// TwinCAT 3 PLC project MC3_Multi_IPC2
// ProgramVersion: 3.1.4026.13
// libraries:
//   Tc2_Standard, * (Beckhoff Automation GmbH)
//   Tc2_System, * (Beckhoff Automation GmbH)
//   Tc3_EventLogger, * (Beckhoff Automation GmbH)
//   Tc3_Mc3PlanarMotion, * (Beckhoff Automation GmbH)
//   Tc3_Module, * (Beckhoff Automation GmbH)
//   Tc3_Physics, * (Beckhoff Automation GmbH)
//   Tc3_XL_Motion, * (Beckhoff Automation GmbH)
//   Tc3_XtsInterface,newest,Beckhoff Automation GmbH
// project tree:
//   DUTs/ E_EcState.TcDUT (not stored), E_MergeMode.TcDUT, E_MergeType.TcDUT, E_SwitchOpMode.TcDUT, E_TrackNum.TcDUT, MoverSort.TcDUT, ST_Color_Code.TcDUT (not stored), ST_DataExchange.TcDUT, ST_DivertConfig.TcDUT (not stored), ST_ExchangeData.TcDUT, ST_ExpMoverStatus.TcDUT, ST_MergeConfig.TcDUT (not stored), ST_MoverConfig.TcDUT (not stored), ST_PlanarTrackConfig.TcDUT, ST_SectorConfig.TcDUT, ST_ShortcutConfig.TcDUT, ST_StaticSectorStatus.TcDUT, ST_SwitchConfig.TcDUT (not stored), ST_SwitchStatus.TcDUT, ST_TrackConfig.TcDUT
//   / FB_XtsDataLoggerForController.TcPOU (excluded from build), PlcTask.TcTTO
//   GVLs/ GVL_DataExchange.TcGVL, GVL_MC.TcGVL
//   POUs/ MAIN_S2.TcPOU
//   XlMover/DUTs/ DUT.TcDUT
//   XlMover/ITFs/ I_Mover.TcIO
//   XlMover/POUs/ FB_Mover.TcPOU, F_GetTrackEnum.TcPOU
// (motion and I/O tree: see PLC project saftyplc)
// real-time tasks:
//   TASK XTS Task: cycle T#500us, priority 1, ADS port 350
//   TASK Job Task: cycle default, priority 32
//   TASK MC-Task (MET): cycle T#2ms, priority 3, ADS port 521
//   TASK MC-Task (MPT): cycle T#10ms, priority 8, ADS port 531
//   TASK PlcTask: cycle T#500us, priority 20, ADS port 351
// variable links:
//   MC3_Multi_IPC2/MC3_Multi_IPC2 Instance <-> Device 2 (EtherCAT Automation Protocol)/Box 29 (Subscriber)
//     PlcTask Inputs/GVL_DataExchange.Dynamics <-> Command/Inputs/VarData/Dynamics
//   MC3_Multi_IPC2/MC3_Multi_IPC2 Instance <-> MC Project IPC2/Axes/MC_Mover 01 IPC2
//     PlcTask Inputs/GVL_MC.fbMover[1].fbPlanarMover.MCTOPLC/ACT <-> McToPlc/ACT
//     PlcTask Inputs/GVL_MC.fbMover[1].fbPlanarMover.MCTOPLC/COORDMODE <-> McToPlc/COORDMODE
//     PlcTask Inputs/GVL_MC.fbMover[1].fbPlanarMover.MCTOPLC/SET <-> McToPlc/SET
//     PlcTask Inputs/GVL_MC.fbMover[1].fbPlanarMover.MCTOPLC/SETONTRACK <-> McToPlc/SETONTRACK
//     PlcTask Inputs/GVL_MC.fbMover[1].fbPlanarMover.MCTOPLC/STD <-> McToPlc/STD
//     PlcTask Outputs/GVL_MC.fbMover[1].fbPlanarMover.PLCTOMC/STD <-> PlcToMc/STD
//   MC3_Multi_IPC2/MC3_Multi_IPC2 Instance <-> MC Project IPC2/Axes/MC_Mover 02 IPC2
//     PlcTask Inputs/GVL_MC.fbMover[2].fbPlanarMover.MCTOPLC/ACT <-> McToPlc/ACT
//     PlcTask Inputs/GVL_MC.fbMover[2].fbPlanarMover.MCTOPLC/COORDMODE <-> McToPlc/COORDMODE
//     PlcTask Inputs/GVL_MC.fbMover[2].fbPlanarMover.MCTOPLC/SET <-> McToPlc/SET
//     PlcTask Inputs/GVL_MC.fbMover[2].fbPlanarMover.MCTOPLC/SETONTRACK <-> McToPlc/SETONTRACK
//     PlcTask Inputs/GVL_MC.fbMover[2].fbPlanarMover.MCTOPLC/STD <-> McToPlc/STD
//     PlcTask Outputs/GVL_MC.fbMover[2].fbPlanarMover.PLCTOMC/STD <-> PlcToMc/STD
//   MC3_Multi_IPC2/MC3_Multi_IPC2 Instance <-> MC Project IPC2/Axes/MC_Mover 03 IPC2
//     PlcTask Inputs/GVL_MC.fbMover[3].fbPlanarMover.MCTOPLC/ACT <-> McToPlc/ACT
//     PlcTask Inputs/GVL_MC.fbMover[3].fbPlanarMover.MCTOPLC/COORDMODE <-> McToPlc/COORDMODE
//     PlcTask Inputs/GVL_MC.fbMover[3].fbPlanarMover.MCTOPLC/SET <-> McToPlc/SET
//     PlcTask Inputs/GVL_MC.fbMover[3].fbPlanarMover.MCTOPLC/SETONTRACK <-> McToPlc/SETONTRACK
//     PlcTask Inputs/GVL_MC.fbMover[3].fbPlanarMover.MCTOPLC/STD <-> McToPlc/STD
//     PlcTask Outputs/GVL_MC.fbMover[3].fbPlanarMover.PLCTOMC/STD <-> PlcToMc/STD
//   MC3_Multi_IPC2/MC3_Multi_IPC2 Instance <-> MC Project IPC2/Axes/MC_Mover 04 IPC2
//     PlcTask Inputs/GVL_MC.fbMover[4].fbPlanarMover.MCTOPLC/ACT <-> McToPlc/ACT
//     PlcTask Inputs/GVL_MC.fbMover[4].fbPlanarMover.MCTOPLC/COORDMODE <-> McToPlc/COORDMODE
//     PlcTask Inputs/GVL_MC.fbMover[4].fbPlanarMover.MCTOPLC/SET <-> McToPlc/SET
//     PlcTask Inputs/GVL_MC.fbMover[4].fbPlanarMover.MCTOPLC/SETONTRACK <-> McToPlc/SETONTRACK
//     PlcTask Inputs/GVL_MC.fbMover[4].fbPlanarMover.MCTOPLC/STD <-> McToPlc/STD
//     PlcTask Outputs/GVL_MC.fbMover[4].fbPlanarMover.PLCTOMC/STD <-> PlcToMc/STD
//   MC3_Multi_IPC2/MC3_Multi_IPC2 Instance <-> MC Project IPC2/Axes/MC_Mover 05 IPC2
//     PlcTask Inputs/GVL_MC.fbMover[5].fbPlanarMover.MCTOPLC/ACT <-> McToPlc/ACT
//     PlcTask Inputs/GVL_MC.fbMover[5].fbPlanarMover.MCTOPLC/COORDMODE <-> McToPlc/COORDMODE
//     PlcTask Inputs/GVL_MC.fbMover[5].fbPlanarMover.MCTOPLC/SET <-> McToPlc/SET
//     PlcTask Inputs/GVL_MC.fbMover[5].fbPlanarMover.MCTOPLC/SETONTRACK <-> McToPlc/SETONTRACK
//     PlcTask Inputs/GVL_MC.fbMover[5].fbPlanarMover.MCTOPLC/STD <-> McToPlc/STD
//     PlcTask Outputs/GVL_MC.fbMover[5].fbPlanarMover.PLCTOMC/STD <-> PlcToMc/STD
//   MC3_Multi_IPC2/MC3_Multi_IPC2 Instance <-> MC Project IPC2/Axes/MC_Mover 06 IPC2
//     PlcTask Inputs/GVL_MC.fbMover[6].fbPlanarMover.MCTOPLC/ACT <-> McToPlc/ACT
//     PlcTask Inputs/GVL_MC.fbMover[6].fbPlanarMover.MCTOPLC/COORDMODE <-> McToPlc/COORDMODE
//     PlcTask Inputs/GVL_MC.fbMover[6].fbPlanarMover.MCTOPLC/SET <-> McToPlc/SET
//     PlcTask Inputs/GVL_MC.fbMover[6].fbPlanarMover.MCTOPLC/SETONTRACK <-> McToPlc/SETONTRACK
//     PlcTask Inputs/GVL_MC.fbMover[6].fbPlanarMover.MCTOPLC/STD <-> McToPlc/STD
//     PlcTask Outputs/GVL_MC.fbMover[6].fbPlanarMover.PLCTOMC/STD <-> PlcToMc/STD
//   MC3_Multi_IPC2/MC3_Multi_IPC2 Instance <-> MC Project IPC2/Axes/MC_Mover 07 IPC2
//     PlcTask Inputs/GVL_MC.fbMover[7].fbPlanarMover.MCTOPLC/ACT <-> McToPlc/ACT
//     PlcTask Inputs/GVL_MC.fbMover[7].fbPlanarMover.MCTOPLC/COORDMODE <-> McToPlc/COORDMODE
//     PlcTask Inputs/GVL_MC.fbMover[7].fbPlanarMover.MCTOPLC/SET <-> McToPlc/SET
//     PlcTask Inputs/GVL_MC.fbMover[7].fbPlanarMover.MCTOPLC/SETONTRACK <-> McToPlc/SETONTRACK
//     PlcTask Inputs/GVL_MC.fbMover[7].fbPlanarMover.MCTOPLC/STD <-> McToPlc/STD
//     PlcTask Outputs/GVL_MC.fbMover[7].fbPlanarMover.PLCTOMC/STD <-> PlcToMc/STD
//   MC3_Multi_IPC2/MC3_Multi_IPC2 Instance <-> MC Project IPC2/Axes/MC_Mover 08 IPC2
//     PlcTask Inputs/GVL_MC.fbMover[8].fbPlanarMover.MCTOPLC/ACT <-> McToPlc/ACT
//     PlcTask Inputs/GVL_MC.fbMover[8].fbPlanarMover.MCTOPLC/COORDMODE <-> McToPlc/COORDMODE
//     PlcTask Inputs/GVL_MC.fbMover[8].fbPlanarMover.MCTOPLC/SET <-> McToPlc/SET
//     PlcTask Inputs/GVL_MC.fbMover[8].fbPlanarMover.MCTOPLC/SETONTRACK <-> McToPlc/SETONTRACK
//     PlcTask Inputs/GVL_MC.fbMover[8].fbPlanarMover.MCTOPLC/STD <-> McToPlc/STD
//     PlcTask Outputs/GVL_MC.fbMover[8].fbPlanarMover.PLCTOMC/STD <-> PlcToMc/STD
//   MC3_Multi_IPC2/MC3_Multi_IPC2 Instance <-> MC Project IPC2/Axes/MC_Mover 09 IPC2
//     PlcTask Inputs/GVL_MC.fbMover[9].fbPlanarMover.MCTOPLC/ACT <-> McToPlc/ACT
//     PlcTask Inputs/GVL_MC.fbMover[9].fbPlanarMover.MCTOPLC/COORDMODE <-> McToPlc/COORDMODE
//     PlcTask Inputs/GVL_MC.fbMover[9].fbPlanarMover.MCTOPLC/SET <-> McToPlc/SET
//     PlcTask Inputs/GVL_MC.fbMover[9].fbPlanarMover.MCTOPLC/SETONTRACK <-> McToPlc/SETONTRACK
//     PlcTask Inputs/GVL_MC.fbMover[9].fbPlanarMover.MCTOPLC/STD <-> McToPlc/STD
//     PlcTask Outputs/GVL_MC.fbMover[9].fbPlanarMover.PLCTOMC/STD <-> PlcToMc/STD
//   MC3_Multi_IPC2/MC3_Multi_IPC2 Instance <-> MC Project IPC2/Axes/MC_Mover 10 IPC2
//     PlcTask Inputs/GVL_MC.fbMover[10].fbPlanarMover.MCTOPLC/ACT <-> McToPlc/ACT
//     PlcTask Inputs/GVL_MC.fbMover[10].fbPlanarMover.MCTOPLC/COORDMODE <-> McToPlc/COORDMODE
//     PlcTask Inputs/GVL_MC.fbMover[10].fbPlanarMover.MCTOPLC/SET <-> McToPlc/SET
//     PlcTask Inputs/GVL_MC.fbMover[10].fbPlanarMover.MCTOPLC/SETONTRACK <-> McToPlc/SETONTRACK
//     PlcTask Inputs/GVL_MC.fbMover[10].fbPlanarMover.MCTOPLC/STD <-> McToPlc/STD
//     PlcTask Outputs/GVL_MC.fbMover[10].fbPlanarMover.PLCTOMC/STD <-> PlcToMc/STD
//   MC3_Multi_IPC2/MC3_Multi_IPC2 Instance <-> MC Project IPC2/Axes/MC_Mover 11 IPC2
//     PlcTask Inputs/GVL_MC.fbMover[11].fbPlanarMover.MCTOPLC/ACT <-> McToPlc/ACT
//     PlcTask Inputs/GVL_MC.fbMover[11].fbPlanarMover.MCTOPLC/COORDMODE <-> McToPlc/COORDMODE
//     PlcTask Inputs/GVL_MC.fbMover[11].fbPlanarMover.MCTOPLC/SET <-> McToPlc/SET
//     PlcTask Inputs/GVL_MC.fbMover[11].fbPlanarMover.MCTOPLC/SETONTRACK <-> McToPlc/SETONTRACK
//     PlcTask Inputs/GVL_MC.fbMover[11].fbPlanarMover.MCTOPLC/STD <-> McToPlc/STD
//     PlcTask Outputs/GVL_MC.fbMover[11].fbPlanarMover.PLCTOMC/STD <-> PlcToMc/STD
//   MC3_Multi_IPC2/MC3_Multi_IPC2 Instance <-> MC Project IPC2/Axes/MC_Mover 12 IPC2
//     PlcTask Inputs/GVL_MC.fbMover[12].fbPlanarMover.MCTOPLC/ACT <-> McToPlc/ACT
//     PlcTask Inputs/GVL_MC.fbMover[12].fbPlanarMover.MCTOPLC/COORDMODE <-> McToPlc/COORDMODE
//     PlcTask Inputs/GVL_MC.fbMover[12].fbPlanarMover.MCTOPLC/SET <-> McToPlc/SET
//     PlcTask Inputs/GVL_MC.fbMover[12].fbPlanarMover.MCTOPLC/SETONTRACK <-> McToPlc/SETONTRACK
//     PlcTask Inputs/GVL_MC.fbMover[12].fbPlanarMover.MCTOPLC/STD <-> McToPlc/STD
//     PlcTask Outputs/GVL_MC.fbMover[12].fbPlanarMover.PLCTOMC/STD <-> PlcToMc/STD
//   MC3_Multi_IPC2/MC3_Multi_IPC2 Instance <-> MC Project IPC2/Groups/IPC 2 In Connection
//     PlcTask Inputs/GVL_MC.EnterSystem.MCTOPLC_STD <-> McToPlc/STD
//   MC3_Multi_IPC2/MC3_Multi_IPC2 Instance <-> MC Project IPC2/Groups/IPC 2 Out Connection
//     PlcTask Inputs/GVL_MC.ExitSystem.MCTOPLC_STD <-> McToPlc/STD
//   MC3_Multi_IPC2/MC3_Multi_IPC2 Instance <-> MC Project IPC2/Groups/McTrack1
//     PlcTask Inputs/GVL_MC.aMcTracks[1].MCTOPLC_STD <-> McToPlc/STD

CONFIGURATION MC3_Multi_IPC2
    RESOURCE PLC ON TwinCAT3
        TASK PlcTask(INTERVAL := T#500us, PRIORITY := 20);
        PROGRAM MAIN_S2 WITH PlcTask : MAIN_S2;
    END_RESOURCE
END_CONFIGURATION

// ---- DUTs/E_MergeMode.TcDUT
{attribute 'qualified_only'}
{attribute 'strict'}
TYPE E_MergeMode :
(
	BlockedWait := 0,
	Follow := 1,
	Lead := 2
);
END_TYPE

// ---- DUTs/E_MergeType.TcDUT
{attribute 'qualified_only'}
{attribute 'strict'}
TYPE E_MergeType :
(
	NoSlowdown := 0,
	StartFromMergeWaitStatic := 1,
	Decelerating := 2 
);
END_TYPE

// ---- DUTs/E_SwitchOpMode.TcDUT
{attribute 'qualified_only'}
//{attribute 'strict'}
TYPE E_SwitchOpMode :
(
  DivertSpecifiedCount	:= 0,
  DivertAll	:= 1
);
END_TYPE

// ---- DUTs/E_TrackNum.TcDUT
TYPE E_TrackNum :
{attribute 'qualified_only'}
{attribute 'strict'}
	(
	MainStart 	:= 1,	
	Big 		:= 1,
	Small 		:= 1,
	MainEnd		:= 1);	
END_TYPE

// ---- DUTs/MoverSort.TcDUT
TYPE MoverSort :
STRUCT
	MoverNumber : UDINT;
	TrackID : PlanarTrackOTCID;
	MoverPos : LREAL;
END_STRUCT
END_TYPE

// ---- DUTs/ST_DataExchange.TcDUT
TYPE ST_DataExchange : 
	STRUCT
	
		Dynamics : ST_Dynamics;
		Reset : BOOL;
		Run : BOOL;
		SafetyInRun : BOOL;
		{attribute 'hide'}
		_reserved1 : ARRAY [1..5] OF USINT;
	END_STRUCT
END_TYPE

// ---- DUTs/ST_ExchangeData.TcDUT
TYPE ST_ExchangeData :
STRUCT
END_STRUCT
END_TYPE

// ---- DUTs/ST_ExpMoverStatus.TcDUT
TYPE ST_ExpMoverStatus :
STRUCT
	XtsBaseRefData						: REFERENCE TO Tc3_XTS_Utility.ST_PositionInfo;
	HasInterference						: BOOL;
	TrackSectorBndryHeadF			: LREAL;
	TrackSectorBndryTailF			: LREAL;
	TrackSectorCenterHead			: LREAL;
	TrackSectorCenterTail			: LREAL;
	TrackSectorBndryHeadR			: LREAL;
	TrackSectorBndryTailR			: LREAL;
	PartSectorBndryHeadF			: LREAL;
	PartSectorBndryTailF			: LREAL;
	PartSectorCenterHead			: LREAL;
	PartSectorCenterTail			: LREAL;
	PartSectorBndryHeadR			: LREAL;
	PartSectorBndryTailR			: LREAL;
	XtsAdjustedData						: Tc3_XTS_Utility.ST_PositionInfo;
END_STRUCT
END_TYPE

// ---- DUTs/ST_PlanarTrackConfig.TcDUT
TYPE ST_PlanarTrackConfig :
STRUCT
	TrackIndex					: E_TrackNum;
	MCTrack						: CDT_MCTOPLC_PLANAR_TRACK;
END_STRUCT
END_TYPE

// ---- DUTs/ST_SectorConfig.TcDUT
TYPE ST_SectorConfig :
STRUCT
	TrackObjectId			: OTCID;
	PartObjectId	    : OTCID;
	PartObjectIdEnt	    : OTCID;
	PartObjectIdExit    : OTCID;	
	PartSectorStartPosn				: LREAL;
	PartSectorEndPosn				: LREAL;
	TrackSectorStartPosn				: LREAL;
	TrackSectorEndPosn				: LREAL;
	SectorSpansBoundary		: BOOL;
END_STRUCT
END_TYPE

// ---- DUTs/ST_ShortcutConfig.TcDUT
TYPE ST_ShortcutConfig :
STRUCT
	TestPowerMat  						: BOOL;
END_STRUCT
END_TYPE

// ---- DUTs/ST_StaticSectorStatus.TcDUT
TYPE ST_StaticSectorStatus :
STRUCT
	MoverIsOnSector			: BOOL;
	MoverCountOnSector		: UDINT;
	MoverEnteredSector		: Tc2_Standard.R_TRIG;
	MoverExitedSector		: Tc2_Standard.F_TRIG;
	SectorLength				: LREAL;
	MoverDistanceFromEnd	: LREAL;
END_STRUCT
END_TYPE

// ---- DUTs/ST_SwitchStatus.TcDUT
TYPE ST_SwitchStatus :
STRUCT
 	MagnetValue		        AT%Q* 	: INT;
	MagnetEnabled     	        	: BOOL;
    CurrentOutputActual             : LREAL;
    CurrentTheoreticalEstimation    : LREAL;
    CurrentOutputMax                : LREAL;
    PosnCurrentCoeff                : LREAL;
	ShuttleCountAtDivertTrig		: UDINT;
	ShuttleQueueCount				: UDINT;
	ShuttleCountOnShortcut			: UDINT;
END_STRUCT
END_TYPE

// ---- DUTs/ST_TrackConfig.TcDUT
TYPE ST_TrackConfig :
STRUCT
	TargetPosnBeforeTrackEnd					: LREAL := 100;
	StopPosPowermat										: LREAL := 7611; // Track Ref; Part Ref ~ 3750 (mm)
	MergeWaitFinishDistance 					: LREAL := 1570;
	MergeWaitAccelDistance						: LREAL; // distance to achieve v_max on the shortcut HD motor region
	ShortcutHDRegionDistance					: LREAL := 2000;
	ShortcutShuttleFullyInPosn 				: LREAL := 1500; // Part Reference (not Track)
	ExpMoverLength										: LREAL := 1200; // roughly 2X SHUTTLE_LENGTH
	MaxLagDistance										: LREAL := 100;
	MergeCollisionRegionDeltaFromL		: LREAL := 2800; // 1715
	MergeCollisionAdvance				: LREAL := 200;
END_STRUCT
END_TYPE

// ---- XlMover/DUTs/DUT.TcDUT
TYPE ST_XtsCommandFeedback :
STRUCT
		(* Returns wether the execution of the method is done. *)
		IsDone : BOOL;
		(* Returns wether the execution of the method is busy. *)
		IsBusy : BOOL;
		(* Returns wether the execution of the method is busy. *)
		HasError : BOOL;
		(* Returns the HRESULT to the call. *)
		{attribute 'GUID' := '18071995-0000-0000-0000-000000000019'}
		{attribute 'GlobalType'}
		HRESULT : GLOBAL.HRESULT;
	END_STRUCT
END_TYPE

// ---- GVLs/GVL_DataExchange.TcGVL
{attribute 'qualified_only'}
VAR_GLOBAL
	Dynamics AT%I*: ST_Dynamics;
		
	aMoverInfos : ARRAY[1..nNumMovers] OF ST_MoverInfo;
END_VAR

// ---- GVLs/GVL_MC.TcGVL

VAR_GLOBAL CONSTANT
	nNumMovers					: UINT := 12;
	nNumTracks					: UINT := 1;
	XtsShortcutOid				: otcid := 16#010100B0 ;
	XtsOutterLoopOid 			: otcid := 16#01010300;
END_VAR

VAR_GLOBAL PERSISTENT
	nNumActiveMovers 			: UINT := 0;
END_VAR

VAR_GLOBAL
	//fbXtsXlMoverUtility 		:	ARRAY[1..nNumMovers] OF FB_XtsXlMoverUtility;
	fbXtsEnvironment			: 	FB_XtsEnvironment;
	ipXtsProcessingUnit			:   I_XtsProcessingUnit1;
	cmdFeedback					: 	XtsCommandFeedback;
	buffer						: 	BYTE;
	
	fbMover						:	ARRAY[1..GVL_MC.nNumMovers] OF FB_Mover;
	iMover						:	ARRAY[1..GVL_MC.nNumMovers] OF I_Mover;
	aDynamics					:  	DynamicConstraint_PathXY;
	Feedback 					:	ARRAY[1..GVL_MC.nNumMovers] OF MC_PlanarFeedback;
	TrackFeedback 				:	ARRAY[1..GVL_MC.nNumTracks] OF MC_PlanarFeedback;
	aMcTracks					:	ARRAY[1..GVL_MC.nNumTracks] OF MC_PlanarTrack;
	ExitSystem 					: 	MC_PlanarTrackConnectionOut;
	EnterSystem 				:	MC_PlanarTrackConnectionIn;
	defaultGap					:	LREAL := 900.0;
END_VAR

// ---- XlMover/ITFs/I_Mover.TcIO

INTERFACE I_Mover

METHOD CycleUpdate : BOOL
VAR_INPUT
END_VAR
END_METHOD

PROPERTY distToEndOfTrack : Lreal
GET
END_GET
END_PROPERTY

METHOD Init : BOOL
VAR_INPUT
	XtsMover:  I_XtsXlMover1;
	XtsProcessingUnit :  I_XtsProcessingUnit1;
END_VAR
END_METHOD

METHOD JoinNearestTrack : BOOL


VAR

END_VAR
END_METHOD

METHOD LeaveSystemAt : BOOL
VAR_INPUT
	ConnectionOut: REFERENCE TO MC_PlanarTrackConnectionOut;	
	gap : LREAL; 	
END_VAR
END_METHOD

METHOD MoveOnTrack : BOOL
VAR_INPUT
	track: REFERENCE TO MC_PlanarTrack;	
	targetPos: LREAL;
	gap : LREAL; 

END_VAR
END_METHOD

PROPERTY MoverStopped : BOOL
GET
END_GET
SET
END_SET
END_PROPERTY

PROPERTY P_Dynamics : REFERENCE TO DynamicConstraint_PathXY;
GET
END_GET
END_PROPERTY

PROPERTY P_IsInitialized : bool
GET
END_GET
END_PROPERTY

PROPERTY P_MoverOTCID : OTCID
GET
END_GET
SET
END_SET
END_PROPERTY

PROPERTY P_PlanarFeedback : REFERENCE TO MC_PlanarFeedback
GET
END_GET
END_PROPERTY

PROPERTY P_PlanarMover :   REFERENCE TO  MC_PlanarMover
GET
END_GET
END_PROPERTY

PROPERTY P_SyncFeedback :  REFERENCE TO MC_PlanarFeedbackGearInPosOnTrackWithMasterMover
GET
END_GET
END_PROPERTY

PROPERTY P_TargetTrack : UDINT
GET
END_GET
SET
END_SET
END_PROPERTY

PROPERTY Rework : BOOL
GET
END_GET
SET
END_SET
END_PROPERTY

METHOD SyncToOtherMover : Bool
VAR_INPUT
	masterSyncPos : LREAL; // Position on the master track
	followerSyncPos : LREAL; // position on the follower track
	PlanarMoverToFollow: REFERENCE TO Tc3_Mc3PlanarMotion.MC_PlanarMover;
	masterTrack : REFERENCE TO Tc3_Mc3PlanarMotion.MC_PlanarTrack; 
	followerTrack : REFERENCE TO Tc3_Mc3PlanarMotion.MC_PlanarTrack; 
	velo :  REFERENCE TO LREAL; 
END_VAR
END_METHOD

METHOD  UpdateXtsTrack
VAR_INPUT
END_VAR
VAR

END_VAR
END_METHOD

PROPERTY XlProcessingUnit : I_XtsProcessingUnit1
GET
END_GET
END_PROPERTY

PROPERTY XtsComFeed : REFERENCE TO  XtsCommandFeedback
GET
END_GET
END_PROPERTY

PROPERTY XtsXlMover :  I_XtsXlMover1
GET
END_GET
END_PROPERTY

END_INTERFACE

// ---- POUs/MAIN_S2.TcPOU
PROGRAM MAIN_S2

VAR
	b110SyncState AT %I* :UINT ;
	b110State AT %I* :UINT;  

	AktiveSystem : BOOL := TRUE;
	bSwitch : BOOL := FALSE;
	nState: UINT;
	CycelCount :ARRAY[1..GVL_MC.nNumMovers] OF INT;
	MoverState :ARRAY[1..GVL_MC.nNumMovers] OF UINT;
	nForCounter ,i: UINT;
	Velo : LREAL := 2000;


	ipXlMover : 	I_XtsXlMover1;


	state AT %Q* : INT := -1;
	arrivedOTCID : OTCID;
	Start :BOOL;
	bAlldone : BOOL;


	test : otcid; 
	XPU_Number : UINT := 1; 	
	
	Short : BOOL;
	
	XtsOutterLoopOid: OTCID ;	
	XtsShortcutOid: OTCID ;

	Init : BOOL ; 
	EndTrack : INT :=E_TrackNum.MainStart ;
 	StartTrack : INT :=E_TrackNum.MainStart ;
	MoverNo : DINT;
	SystemReady: BOOL;
	
	cmdFeedback: Tc3_XtsInterface.XtsCommandFeedback;
	BUFFER: BYTE;
	
	xEapStart AT %I*: BOOL;
	xEAPReset AT %I*: BOOL;
	EtherCATModulesWCState AT %I*: BOOL;
	EhterCATFault: BOOL;
	SyncFault: BOOL;
	
	temp: HRESULT;
	
	haltDynamics : DynamicConstraint_PathXY;
	stMoverConfigSlow	: ST_MoverConfig;
	stMoverConfigNormal : ST_MoverConfig;
	stMoverConfigFast  : ST_MoverConfig;
	stMoverCfgAggressive : ST_MoverConfig;
	stMoverCfgHalt : ST_MoverConfig;
	MoverStopDone : BOOL;
	Fault : BOOL;
	Fp_error : r_trig;
	AllDone : BOOL;
	InitDone  :BOOL;
	PackMovers: BOOL :=TRUE;
END_VAR

// =====================
// Initalize XTS Utility
GVL_MC.fbXtsEnvironment.Init(GVL_MC.cmdFeedback);
IF NOT GVL_MC.cmdFeedback.IsDone THEN
	RETURN;
END_IF

IF  GVL_DataExchange.Dynamics.V = 0 THEN
	stMoverConfigNormal.Velo	:=	1000;
	stMoverConfigNormal.Accel	:=	4000;
	stMoverConfigNormal.Decel	:=	4000;
	stMoverConfigNormal.Jerk	:=	16000;
ELSE
	stMoverConfigNormal.Velo	:=	GVL_DataExchange.Dynamics.v;
	stMoverConfigNormal.Accel	:=	GVL_DataExchange.Dynamics.A;
	stMoverConfigNormal.Decel	:=	GVL_DataExchange.Dynamics.D;
	stMoverConfigNormal.Jerk	:=	GVL_DataExchange.Dynamics.J;
END_IF
haltdynamics.SetValuesVADJ(stMoverConfigNormal.Velo,stMoverConfigNormal.Accel, stMoverConfigNormal.Decel, stMoverConfigNormal.Jerk);

// =====================
GVL_MC.ipXtsProcessingUnit :=  GVL_MC.fbXtsEnvironment.ProcessingUnit(XPU_Number,0);
AllDone := TRUE;
FOR i := 1 TO GVL_MC.nNumMovers DO 
	
	IF NOT InitDone  THEN
		ipXlMover  :=  GVL_MC.fbXtsEnvironment.ProcessingUnit(XPU_Number, 0).XlMover(i, 0);
		AllDone := AllDone AND GVL_MC.fbMover[i].Init(ipXlMover, GVL_MC.ipXtsProcessingUnit); 
	END_IF
	
	
	Fp_error(clk := GVL_MC.fbMover[i].P_PlanarMover.Error AND GVL_MC.fbMover[i].XtsXlMover.GetIsActive(0) AND state = 100);
	IF Fp_error.Q AND FALSE THEN
		state := 140;
		Fault := TRUE;

		ADSLOGSTR(msgCtrlMask:= ADSLOG_MSGTYPE_LOG , msgFmtStr:= 'Mover %s Faulted ' , strArg:= INT_TO_STRING(i));
	ELSE
		Fault := FALSE;
	END_IF
	
	
	GVL_MC.Feedback[i].Update();
	GVL_MC.fbMover[i].CycleUpdate();
	GVL_MC.iMover[i] := GVL_MC.fbMover[i];
	// these are all hard coded and need to be transmitted from PC1 to PC2.  
	IF I = 1 AND PackMovers THEN 
		GVL_MC.fbMover[i].P_Dynamics.SetValuesVADJ(stMoverConfigNormal.Velo-10,stMoverConfigNormal.Accel, stMoverConfigNormal.Decel, stMoverConfigNormal.Jerk);
	ELSE 
		GVL_MC.fbMover[i].P_Dynamics.SetValuesVADJ(stMoverConfigNormal.Velo,stMoverConfigNormal.Accel, stMoverConfigNormal.Decel, stMoverConfigNormal.Jerk);
	END_IF 
	GVL_MC.fbMover[i].P_MoveOnTrackOptions.gap := 900;
	GVL_MC.fbMover[i].P_MoveOnTrackOptions.direction := MC_Direction.mcDirectionPositive;
	GVL_MC.fbMover[i].P_MoveOnTrackOptions.gapMode := MC_GAP_MODE_ON_TRACK.Fast1D;
	GVL_DataExchange.aMoverInfos[i] :=  GVL_MC.fbMover[i].P_MoverInfos;
END_FOR	

IF AllDone THEN
	InitDone := TRUE;
ELSE
	RETURN;
END_IF

FOR i := 1 TO GVL_MC.nNumTracks DO 
	GVL_MC.aMcTracks[i].Update();
	GVL_MC.TrackFeedback[i].Update();
END_FOR	



IF state <99 AND xEAPReset THEN 
	state := 0; 
END_IF

IF state = 99 AND xEAPStart THEN 
	state := 100; 
END_IF

IF EtherCATModulesWCState THEN 
	EhterCATFault := TRUE;
END_IF  

IF b110SyncState <>1 THEN 
	SyncFault := TRUE; 
END_IF



CASE state OF
	0: 
		
		FOR i := 1 TO GVL_MC.nNumTracks DO  
			GVL_MC.aMcTracks[i].Enable(GVL_MC.TrackFeedback[i]);
			state := 1;
		END_FOR
		
	1: 	
		bAlldone := TRUE;
		FOR i := 1 TO GVL_MC.nNumTracks DO  
			bAlldone := bAlldone AND GVL_MC.aMcTracks[i].MCTOPLC_STD.State = MC_PLANAR_STATE.Enabled ;
		END_FOR
			
 		IF bAlldone THEN
			state := 2;
		END_IF

	2:	
		FOR i := 1+GVL_MC.nNumActiveMovers TO GVL_MC.nNumMovers DO  
			GVL_MC.fbMover[i].XlProcessingUnit.XlMover(i,0).SetStartupTrackPosition(0.2,0);	
			GVL_MC.fbMover[i].XlProcessingUnit.XlMover(i,0).SetIsVirtualFeedbackEnabled(1,0);
			GVL_MC.fbMover[i].XlProcessingUnit.XlMover(i,0).TriggerArrive(0);
		END_FOR
		IF  GVL_MC.nNumActiveMovers > 0 THEN
			FOR i :=1  TO GVL_MC.nNumActiveMovers DO 	
				GVL_MC.fbMover[i].XlProcessingUnit.XlMover(i,0).SetIsVirtualFeedbackEnabled(0,0);
			END_FOR 
		END_IF			
		state := 3;
		
	3:
		FOR i := 1 TO GVL_MC.fbXtsEnvironment.ProcessingUnit(1, 0).XlPartCount() DO
			 GVL_MC.fbXtsEnvironment.ProcessingUnit(1, 0).XlPart(i, 0).TriggerReset(0);
		END_FOR
		
		state := 5;
		
	5: 

		
		IF AktiveSystem THEN
			state := 10;
		ELSE
			state := 100;
		END_IF	

	10:
		FOR i := 1 TO GVL_MC.nNumActiveMovers DO
			GVL_MC.fbMover[i].P_PlanarMover.Reset(0);
		END_FOR
		state := 11;
 	11:
		FOR i := 1 TO GVL_MC.nNumActiveMovers DO	
			GVL_MC.fbMover[i].P_PlanarMover.Enable(0);		
		END_FOR
		state := 15;	
	15:
		bAlldone := TRUE;
		FOR i := 1 TO GVL_MC.nNumActiveMovers DO  
			bAlldone := bAlldone AND GVL_MC.fbMover[i].P_PlanarMover.MCTOPLC.STD.State = MC_PLANAR_STATE.Enabled;	
		END_FOR
		
		IF bAlldone THEN
			state := 18;
		END_IF
	18: 
	
		FOR i := 1 TO GVL_MC.nNumActiveMovers DO  
			GVL_MC.fbMover[i].JoinNearestTrack(aMcTracks,nNumTracks );	
		END_FOR
		state := 20;
	
	20:
		bAlldone := TRUE;
		FOR i := 1 TO GVL_MC.nNumActiveMovers DO
			bAlldone := bAlldone AND GVL_MC.fbMover[i].fbPlanarMover.MCTOPLC.STD.CommandMode = MC_PLANAR_MOVER_COMMAND_MODE.OnTrack  ;	
			MoverState[i] := 10;
			
		END_FOR

		IF bAlldone THEN
			state := 99;
		END_IF
		
	100: 
		arrivedOTCID := GVL_MC.EnterSystem.PopFirstMoverInQueue();
		IF arrivedOTCID <> 0 THEN
			FOR i := 1  TO GVL_MC.nNumMovers DO
				IF GVL_MC.fbMover[i].p_MoverOTCID = arrivedOTCID THEN
					MoverState[i] := 0;
				END_IF
			END_FOR
		END_IF
	
		FOR i := 1 TO GVL_MC.nNumMovers DO 
			CASE MoverState[i] OF 
		
			0:
				IF MoverNo <> 0 AND_THEN GVL_MC.fbMover[MoverNo].P_PlanarMover.MCTOPLC.SETONTRACK.TrackOID =  GVL_MC.aMcTracks[E_TrackNum.MainStart].MCTOPLC_STD.TrackOID THEN
					Short := FALSE;
				END_IF
		
				IF GVL_MC.fbMover[i].P_PlanarMover.MCTOPLC.SETONTRACK.SetPos > 100  THEN
					IF NOT short AND bSwitch  THEN
						GVL_MC.fbMover[i].MoveOnTrack(GVL_MC.aMcTracks[E_TrackNum.MainStart],GVL_MC.aMcTracks[E_TrackNum.MainStart].GetLength()/2,GVL_MC.defaultGap);
						MoverNo := i;
						Short := TRUE;
						MoverState[i] := 10;
					ELSE
						GVL_MC.fbMover[i].MoveOnTrack(GVL_MC.aMcTracks[EndTrack],GVL_MC.aMcTracks[EndTrack].GetLength()/2,GVL_MC.defaultGap);			
						MoverState[i] := 10;
					END_IF				
				END_IF
								
			10:
				IF(  GVL_MC.fbMover[i].P_PlanarMover.MCTOPLC.SETONTRACK.SetPos > 500 AND GVL_MC.fbMover[i].P_PlanarMover.MCTOPLC.SETONTRACK.TrackOID <>  GVL_MC.aMcTracks[StartTrack].MCTOPLC_STD.TrackOID) OR GVL_MC.nNumTracks =1 THEN
					GVL_MC.fbMover[i].MoveOnTrack(GVL_MC.aMcTracks[EndTrack],GVL_MC.aMcTracks[EndTrack].GetLength() - 1500,GVL_MC.defaultGap) ;//VElo*0.35);
					MoverState[i] := 11;
				END_IF
			11:	
				//special command no chance to break in time 
				IF  SystemReady  THEN
					GVL_MC.fbMover[i].MoveOnTrack(GVL_MC.aMcTracks[EndTrack],GVL_MC.aMcTracks[EndTrack].GetLength() - 200,GVL_MC.defaultGap);
					//GVL_MC.fbMover[i].MoveOnTrack(GVL_MC.aMcTracks[EndTrack],GVL_MC.aMcTracks[EndTrack].GetLength()-200);
					MoverState[i] := 12;
				END_IF		
			12: IF GVL_MC.fbMover[i].P_PlanarMover.MCTOPLC.SETONTRACK.SetPos > GVL_MC.aMcTracks[EndTrack].GetLength() - 2300 AND 
				(GVL_MC.fbMover[i].P_PlanarMover.MCTOPLC.SETONTRACK.TrackOID = GVL_MC.aMcTracks[EndTrack].MCTOPLC_STD.TrackOID) THEN 
					GVL_MC.fbMover[i].LeaveSystemAt(GVL_MC.ExitSystem, GVL_MC.defaultGap); 
					MoverState[i] := 15; 
				END_IF	
				
			15:
			 	IF GVL_MC.fbMover[i].XlProcessingUnit.XlMover(i,0).GetIsVirtualFeedbackEnabled(0) AND //In some cases the planar mover gots an error, we have to evaluate why
					GVL_MC.fbMover[i].P_PlanarMover.Error THEN
					GVL_MC.fbMover[i].P_PlanarMover.Reset(0);
					MoverState[i] := 16; 
				END_IF
				
			16: 
				GVL_MC.fbMover[i].P_PlanarMover.Disable(0);
				MoverState[i] := 17; 
			END_CASE
		END_FOR
		
		140:
			FOR i := 1 TO GVL_MC.nNumMovers DO  
				GVL_MC.fbMover[i].P_PlanarMover.Halt(GVL_MC.Feedback[i], haltDynamics);
			END_FOR	
			
				state := 145;
			
		145:
			bAllDone := TRUE;
				FOR i := 1 TO GVL_MC.nNumMovers DO  
				IF NOT(GVL_MC.Feedback[i].Done OR GVL_MC.Feedback[i].Error) THEN
					bAllDone := FALSE;
					EXIT;
				END_IF
			END_FOR
			
			IF bAllDone THEN
				state := 150;
			END_IF
		
		//Disable
		150:
			MoverStopDone := TRUE;
			FOR i := 1 TO GVL_MC.nNumMovers DO  
					GVL_MC.fbMover[i].P_PlanarMover.Disable(GVL_MC.Feedback[i]);
			END_FOR
				
			state := 0;
		
	
END_CASE

END_PROGRAM

// ---- XlMover/POUs/FB_Mover.TcPOU
{attribute 'no_assign'}
FUNCTION_BLOCK FB_Mover IMPLEMENTS I_Mover
VAR_INPUT
END_VAR
VAR_OUTPUT
END_VAR
VAR
	_bIsInitialized: BOOL;	

	fbPlanarMover : MC_PlanarMover;
	fbPlanarFeedback: MC_PlanarFeedback;
	trackTrail: MC_PlanarTrackTrail;
	SyncMoverFeedback: Tc3_Mc3PlanarMotion.MC_PlanarFeedbackGearInPosOnTrackWithMasterMover;
	
	_GearInOptions: Tc3_Mc3PlanarMotion.ST_GearInPosOnTrackWithMasterMoverOptions;
	_stMoveOnTrackOptions: ST_MoveOnTrackOptions;
	_stLeaveSystemAtOptions : ST_LeaveSystemAtOptions;
	
	_syncTrail : MC_PlanarTrackTrail;
	
	CmdFeedback :  XtsCommandFeedback;
	ipXtsMover:   I_XtsXlMover1;
	ipXtsProcessingUnit:  I_XtsProcessingUnit1;

	_stMoverInfos : ST_MoverInfo;	
	_stMoverOnTrackInfos : ST_MoverOnTrackInfo;

	_nextMcTrackOid: OTCID;
	_stDynamics: DynamicConstraint_PathXY;
	_TargetTrack : UDINT;
	_ReWork : BOOL;
	_partConfig: UINT;
	_InSync :BOOL; 
	_PositionOnTrack : LREAL;
	_Track : OTCID; 
	_distToEndOfTrack : LREAL;

	fbResult						: FB_TcMessage;
	_ipComObject					: ITComObject;
	PID_OnTrackInfos				: PTCID := 16#05030180;
	bInit 							: BOOL;
END_VAR


METHOD CycleUpdate : BOOL
VAR_INPUT
END_VAR
VAR 
	_trackEnum: e_TrackNum;
END_VAR
IF NOT _bIsInitialized THEN
	RETURN;
END_IF

fbPlanarMover.GetTrackTrailInformation(trackTrail);
_PositionOnTrack := fbPlanarMover.MCTOPLC.SETONTRACK.SetPos;
IF fbPlanarMover.MCTOPLC.SETONTRACK.TrackOID<>0 THEN 
	_Track := fbPlanarMover.MCTOPLC.SETONTRACK.TrackOID;
	_trackEnum := F_GetTrackEnum(fbPlanarMover.MCTOPLC.SETONTRACK.TrackOID); 
	_distToEndOfTrack := GVL_Mc.aMCTracks[_trackEnum].GetLength()-_PositionOnTrack;
END_IF

fbPlanarMover.Update();

_stMoverinfos.MoverOtcid := fbPlanarMover.MCTOPLC.STD.MoverOID ;
_stMoverinfos.IsActive := ipXtsMover.GetIsActive(0);
_stMoverinfos.ActPos :=  ipXtsMover.GetPositionInfo_trackPosition(0);
_stMoverinfos.ActVelo := fbPlanarMover.MCTOPLC.SETONTRACK.SetVelo;
_stMoverinfos.IsVirtuell := ipXtsMover.GetIsVirtualFeedbackEnabled(0);
_stMoverinfos.Positition :=	fbPlanarMover.MCTOPLC.SETONTRACK.SetPos;
_stMoverinfos.Track := fbPlanarMover.MCTOPLC.SETONTRACK.TrackOID;
_stMoverinfos.Error := fbPlanarMover.Error;
_stMoverinfos.ErrorID := fbPlanarMover.ErrorId;
_stMoverinfos.PlanarMoverCommandMode := fbPlanarMover.MCTOPLC.STD.CommandMode;
_stMoverinfos.State :=  fbPlanarMover.MCTOPLC.STD.State;
_stMoverinfos.Gap := _stMoverOnTrackInfos.Gap;
_stMoverinfos.LimitAcc := _stMoverOnTrackInfos.LimitA;
_stMoverinfos.LimitDec := _stMoverOnTrackInfos.LimitD;
_stMoverinfos.LimitJerk := _stMoverOnTrackInfos.LimitJ;
_stMoverinfos.LimitVelo := _stMoverOnTrackInfos.LimitV;
_stMoverinfos.TargetTrackPosition := _stMoverOnTrackInfos.TargetPosition;
_stMoverinfos.TargetTrack := _stMoverOnTrackInfos.TargetTrack;
_stMoverinfos.RemainingDistance := _stMoverOnTrackInfos.Remainingdistance;

fbPlanarFeedback.Update();
SyncMoverFeedback.Update(); 


UpdateXtsTrack();

GetOnTrackInfos();
END_METHOD

PROPERTY distToEndOfTrack : Lreal
GET
distToEndOfTrack := _distToEndOfTrack;
END_GET
END_PROPERTY

METHOD GetComObject : BOOL
VAR_INPUT
	nObjectId: OTCID;
END_VAR
IF FW_ObjMgr_GetObjectInstance(	oid		:= nObjectId, 
								iid		:= TC_GLOBAL_IID_LIST.IID_ITComObject, 
								pipUnk	:= ADR(_ipComObject)) = 0
THEN
	GetComObject := TRUE;
END_IF
END_METHOD

METHOD GetOnTrackInfos : BOOL
VAR
	nData 			: UDINT := SIZEOF(_stMoverOnTrackInfos);
	pData 			: PVOID := ADR(_stMoverOnTrackInfos);
	stEventEntry	: TcEventEntry;
	pstEventEntry	: REFERENCE TO TcEventEntry REF= stEventEntry;
END_VAR
VAR_INST
	hResult : HRESULT;
	bError : BOOL;
END_VAR
bError := FALSE;

IF _ipComObject <> 0 THEN 
	 hResult := 	_ipComObject.TcgetObjPara(		pid := PID_OnTrackInfos,
													nData := nData,
													pData := pData,
													pgp := 0); 	
	IF hResult = 0 THEN
		GetOnTrackInfos := TRUE;
	ELSE
		HRESULTAdsErr_TO_TcEventEntry(hResult,stEventEntry);
		IF NOT fbResult.EqualsToEventEntryEx( stOther := stEventEntry) THEN
			fbResult.CreateEx(stEventEntry, 0);
			fbResult.Send(0);
			fbResult.Release();
		END_IF
		bError := TRUE;
	END_IF							
END_IF
END_METHOD

METHOD Init : BOOL
VAR_INPUT

	XtsMover:   I_XtsXlMover1;
	XtsProcessingUnit :  I_XtsProcessingUnit1;
END_VAR



ipXtsMover:= XtsMover;
ipXtsProcessingUnit :=  XtsProcessingUnit;

_stMoveOnTrackOptions.direction := MC_Direction.mcDirectionPositive;
_stMoveOnTrackOptions.gapMode := MC_GAP_MODE_ON_TRACK.Fast1D;
_stMoveOnTrackOptions.gap:= 800;

_syncTrail.AddTrack(track:= GVL_Mc.aMCTracks[E_TrackNum.Small]); 
_syncTrail.AddTrack(track:= GVL_Mc.aMCTracks[E_TrackNum.MainStart]); 


//_stDynamics.SetValuesVADJ(500, 4000, 4000, 10000);

_bIsInitialized := TRUE;
Init := TRUE;


IF NOT bInit THEN
	IF GetComObject(nObjectId:=fbPlanarMover.MCTOPLC.STD.MoverOID) THEN
		bInit:=TRUE;
	END_IF
	RETURN;
END_IF
END_METHOD

METHOD JoinNearestTrack : BOOL


VAR_INST
	nForCounter: UINT;
	mcTrackOid: OTCID;
	partOid: OTCID;
	cmdFeedback					: 	XtsCommandFeedback;
	objectInfo: PlanarObjectInfo;
END_VAR
partOid := ipXtsMover.GetPositionInfo_partObjectId(cmdFeedback);

IF partOid = 0 THEN
	RETURN;
END_IF

IF cmdFeedback.IsDone THEN
	mcTrackOid := ipXtsProcessingUnit.XlPartWithOid(partOid, cmdFeedback).GetMcTrackOid(cmdFeedback);
	
	FOR nForCounter := 1 TO GVL_MC.nNumTracks DO
		objectInfo := GVL_MC.aMcTracks[nForCounter].GetPlanarObjectInfo();
		IF objectInfo.Id = mcTrackOid THEN
			fbPlanarMover.JoinTrack(fbPlanarFeedback, GVL_MC.aMcTracks[nForCounter], _stDynamics, 0); 
			RETURN;
		END_IF
	END_FOR
END_IF
END_METHOD

METHOD LeaveSystemAt : BOOL
VAR_INPUT
	ConnectionOut: REFERENCE TO MC_PlanarTrackConnectionOut;
	gap : LREAL; 	
END_VAR
_stLeaveSystemAtOptions.gap := gap;
_stLeaveSystemAtOptions.gapMode := MC_GAP_MODE_ON_TRACK.Fast1D; 
_stLeaveSystemAtOptions.dynamicMode :=  MC_DYNAMIC_MODE_ON_TRACK.None;

fbPlanarMover.LeaveSystemAt(fbPlanarFeedback, ConnectionOut,  _stDynamics,_stLeaveSystemAtOptions);
END_METHOD

METHOD MoveOnTrack : BOOL
VAR_INPUT
	track: REFERENCE TO MC_PlanarTrack;	
	targetPos: LREAL;
	gap : LREAL; 
END_VAR
_stMoveonTrackOptions.gap := gap; 

fbPlanarMover.MoveOnTrack(
	commandFeedback:= fbPlanarFeedback, 
	targetTrack:= track, 
	targetPositionOnTrack:= targetPos, 
	constraint:= _stDynamics, 
	options:= _stMoveOnTrackOptions);
END_METHOD

PROPERTY MoverStopped : BOOL
GET
MoverStopped := (fbPlanarMover.MCTOPLC.SETONTRACK.SetVelo < 20);
END_GET
SET
END_SET
END_PROPERTY

PROPERTY P_Dynamics : REFERENCE TO DynamicConstraint_PathXY;
GET

P_Dynamics REF= _stDynamics;
END_GET
SET // PUBLIC
_stDynamics := P_Dynamics;
END_SET
END_PROPERTY

PROPERTY P_IsInitialized : bool
GET
P_IsInitialized := _bIsInitialized;
END_GET
END_PROPERTY

PROPERTY P_MoveOnTrackOptions  : REFERENCE TO  ST_MoveOnTrackOptions
GET
P_MoveOnTrackOptions REF= _stMoveOnTrackOptions;
END_GET
END_PROPERTY

PROPERTY P_MoverInfos : REFERENCE TO ST_MoverInfo
GET
P_MoverInfos  REF= _stMoverInfos;
END_GET
END_PROPERTY

PROPERTY p_MoverOTCID : OTCID
GET
p_MoverOTCID := fbPlanarMover.MCTOPLC.STD.MoverOID;
END_GET
SET
END_SET
END_PROPERTY

PROPERTY P_PlanarFeedback : REFERENCE TO MC_PlanarFeedback
GET
P_PlanarFeedback REF= fbPlanarFeedback;
END_GET
END_PROPERTY

PROPERTY P_PlanarMover :   REFERENCE TO  MC_PlanarMover
GET
P_PlanarMover REF= fbPlanarMover;
END_GET
END_PROPERTY

PROPERTY P_SyncFeedback :  REFERENCE TO MC_PlanarFeedbackGearInPosOnTrackWithMasterMover
GET
P_SyncFeedback REF= SyncMoverFeedback;
END_GET
END_PROPERTY

PROPERTY P_TargetTrack : UDINT
GET
P_TargetTrack := _TargetTrack ;
END_GET
SET
_TargetTrack := P_TargetTrack;
END_SET
END_PROPERTY

PROPERTY Rework : BOOL
GET
Rework := _Rework;
END_GET
SET
_Rework := Rework;
END_SET
END_PROPERTY

METHOD SyncToOtherMover : BOOL
VAR_INPUT
	masterSyncPos : LREAL; // Position on the master track
	followerSyncPos : LREAL; // position on the follower track
	PlanarMoverToFollow: REFERENCE TO Tc3_Mc3PlanarMotion.MC_PlanarMover;
	masterTrack : REFERENCE TO Tc3_Mc3PlanarMotion.MC_PlanarTrack; 
	followerTrack : REFERENCE TO Tc3_Mc3PlanarMotion.MC_PlanarTrack; 
	velo : REFERENCE TO LREAL; 
END_VAR

VAR
	trail: Tc3_Mc3PlanarMotion.MC_PlanarTrackTrail;

END_VAR
_GearInOptions.allowedSlaveSyncDirections := MC_SYNC_DIRECTIONS.Positive; 
_GearInOptions.directionMasterSyncPosition := MC_DIRECTION.mcDirectionNonModulo; 
_GearInOptions.directionSlaveSyncPosition := MC_DIRECTION.mcDirectionNonModulo;  
_GearInOptions.followMover := FALSE; 
_GearInOptions.gap := 0; // elimnate gap funciton 
_GearInOptions.inSyncToleranceDistance :=0; 
_GearInOptions.moduloToleranceMasterSyncPosition := 0; 
_GearInOptions.moduloToleranceSlaveSyncPosition := 0;  
_stDynamics.V := velo; 

fbPlanarMover.GearInPosOnTrackWithMasterMover(
	commandFeedback:=  SyncMoverFeedback , 
	masterMover:= PlanarMoverToFollow , 
	trackTrail:= _syncTrail, // may need to give a trail maybe not
	masterSyncPosition:= masterSyncPos, 
	masterSyncPositionTrack:= MasterTrack , 
	slaveSyncPosition:= followerSyncPos, 
	slaveSyncPositionTrack:= followerTrack, 
	constraint:=_stDynamics , 
	options:=_GearInOptions );
END_METHOD

METHOD PUBLIC UpdateXtsTrack
VAR_INPUT
END_VAR
VAR_STAT
	nTrackCount: UINT;
	oid1: OTCID;
	oid2: OTCID;
	
	nForCounter: UINT;
	nPartConfigCount: UINT;
	
	partConfig1: OTCID;
	partConfig2: OTCID;
	
	mcTrackOid1: OTCID;
	mcTrackOid2: OTCID;
	trackOid: OTCID;
	
	nTrackTrailCount: UDINT;
	actTrackOid: OTCID;
	nIndexInTrail: UDINT;
END_VAR
nTrackTrailCount := trackTrail.TrackCount;
actTrackOid := fbPlanarMover.MCTOPLC.SETONTRACK.TrackOID;

IF nTrackTrailCount <= 1 THEN
	RETURN;
END_IF

FOR nForCounter := 1 TO UDINT_TO_UINT(nTrackTrailCount) DO
	oid1 := trackTrail.GetTrackOidAt(nForCounter);
	IF oid1 = actTrackOid THEN
		IF nForCounter < nTrackTrailCount THEN
			oid2 := trackTrail.GetTrackOidAt(nForCounter + 1);
			EXIT;
		ELSE
			RETURN; //last one ine track trail
		END_IF
	END_IF
END_FOR

IF oid2 = _nextMcTrackOid AND   ipXtsMover.GetPositionInfo_partPosition(CmdFeedback) < 600THEN //no change
	RETURN;
END_IF

nTrackCount := ipXtsProcessingUnit.TrackCount();

FOR nForCounter := 1 TO nTrackCount DO
	nPartConfigCount := ipXtsProcessingUnit.Track(nForCounter, CmdFeedback).PartConfigCount(); 
	
	IF nPartConfigCount >= 2  THEN
		partConfig1 := ipXtsProcessingUnit.Track(nForCounter, CmdFeedback).GetPartConfigOidAt(1, 0);
		partConfig2 := ipXtsProcessingUnit.Track(nForCounter, CmdFeedback).GetPartConfigOidAt(2, 0);
//
		
		IF partConfig1 = 0 OR partConfig2 = 0 THEN
			CONTINUE;
		END_IF
		
		mcTrackOid1 := ipXtsProcessingUnit.XlPartWithOid(partConfig1, CmdFeedback).GetMcTrackOid(0);
		mcTrackOid2 := ipXtsProcessingUnit.XlPartWithOid(partConfig2, CmdFeedback).GetMcTrackOid(0);
		IF mcTrackOid1 = oid1 AND mcTrackOid2 = oid2   THEN
			trackOid := ipXtsProcessingUnit.Track(nForCounter, CmdFeedback).GetObjectId();
			ipXtsMover.SetActiveTrackObjectId(trackOid, CmdFeedback);
			
			IF CmdFeedback.IsDone THEN
				_nextMcTrackOid := oid2;
			END_IF
			
			RETURN;
		END_IF
	END_IF
END_FOR
END_METHOD

PROPERTY XlProcessingUnit : I_XtsProcessingUnit1
GET
XlProcessingUnit := ipXtsProcessingUnit;
END_GET
END_PROPERTY

PROPERTY XtsComFeed : REFERENCE TO  XtsCommandFeedback
GET
XtsComFeed REF= CmdFeedback;
END_GET
END_PROPERTY

PROPERTY XtsXlMover : I_XtsXlMover1
GET
XtsXlMover := ipXtsMover;
END_GET
END_PROPERTY

END_FUNCTION_BLOCK

// ---- XlMover/POUs/F_GetTrackEnum.TcPOU
FUNCTION F_GetTrackEnum : E_TrackNum
VAR_INPUT
	Track : otcid;
END_VAR
VAR
END_VAR

IF GVL_Mc.aMCTracks[E_TrackNum.MainStart].MCTOPLC_STD.TrackOID = track THEN 
                F_GetTrackEnum := E_TrackNum.MainStart; 
ELSIF 
                GVL_Mc.aMCTracks[E_TrackNum.MainEnd].MCTOPLC_STD.TrackOID = track THEN 
                F_GetTrackEnum := E_TrackNum.MainEnd; 
ELSIF 
                GVL_Mc.aMCtracks[E_TrackNum.Big].MCTOPLC_STD.TrackOID = track THEN 
                F_GetTrackEnum := E_TrackNum.Big;
ELSIF 
                GVL_Mc.aMCtracks[E_TrackNum.Small].MCTOPLC_STD.TrackOID = track THEN 
                F_GetTrackEnum := E_TrackNum.Small; 
 
END_IF

END_FUNCTION

// ---- FB_XtsDataLoggerForController.TcPOU
FUNCTION_BLOCK FB_XtsDataLoggerForController
VAR_INPUT
	iXtsEnv 			: I_TcIoXtsEnvironment; 
	nNumOfMovers		: UINT; 
END_VAR
VAR_OUTPUT
	bReady				: BOOL := FALSE;
	nErrorID			: HRESULT; 
END_VAR

VAR PERSISTENT
	PersistentRollerID : ARRAY[1..nNumMovers] OF INT;
	PersistentRollerExchangeDate : ARRAY[1..nNumMovers] OF STRING;
END_VAR


VAR
{region "Background Handling"}
	//During Init() all Pointer Addresses are stored in this struct
	stPointerAddresses: ARRAY[1..nNumMovers] OF ST_XtsControllerPointer;
	ControllerOID		: ARRAY [1..nNumMovers] OF OTCID; 
{endregion}
	
{region "Data Logging Application"}	
	nMover			: INT;

	{attribute 'TcAnalytics'}
	aMoverData				: ARRAY[1..nNumMovers] OF ST_MoverData;
	{attribute 'TcAnalytics'}
	aMoverDataReduced		: ARRAY[1..nNumMovers] OF	ST_MoverDataReduced;

{endregion}
	
END_VAR

//wait until XTS Application is ready before anything else is done
IF  iXtsEnv <> 0 THEN
	IF iXtsEnv.P_IsInitialized THEN
		// Initialize the Logger FB
		IF NOT bReady  THEN
			bReady:= Init(); 
			RETURN; 
		ELSE 
			//once everything is initialized, start reading data
			ccl_UpdateMoverData(); 
		END_IF 	
	END_IF 
END_IF

METHOD ccl_UpdateMoverData : BOOL
VAR_INPUT
END_VAR

// -------------------------------------- Retrieve and compute mover data -----------------------------------------
FOR nMover:=1 TO nNumOfMovers DO
	// ***************************************Part 1: assign mover data to an array *****************************//
	//1. Act Current
	aMoverData[nMover].SetCurrent := stPointerAddresses[nMover].SetCurrentPointer ^; 
	//3. Aktuelle ungefilterte Modulo Istposition			
	aMoverData[nMover].ActHwPosModulo := stPointerAddresses[nMover].ActHwPosModuloPointer^;
	//4. actFollowingError (gefilterter Schleppfehler in 0.1 micrometer)
	aMoverData[nMover].ActPosError := stPointerAddresses[nMover].ActPosErrorPointer^;
	//5.  Set velocityItp
	aMoverData[nMover].SetVeloItp := stPointerAddresses[nMover].SetVeloItpPointer^;
	//6. Set AccItp
	aMoverData[nMover].SetAccItp := stPointerAddresses[nMover].SetAccItpPointer^;
	//7. ActVelo
	aMoverData[nMover].actVelo := stPointerAddresses[nMover].ActVeloPointer^;
	//8. Roller ID
	aMoverData[nMover].RollerID := PersistentRollerID[nMover]; 

	//*************************************** Part 2: assign mover data for reduced set of variables ********************//

	//1. Actual current command
	aMoverDataReduced[nMover].SetCurrent := stPointerAddresses[nMover].SetCurrentPointer^; 
	//3. Aktuelle ungefilterte Modulo Istposition			
	aMoverDataReduced[nMover].ActHwPosModulo := stPointerAddresses[nMover].ActHwPosModuloPointer^;
	//8.  Set velocityItp
	aMoverDataReduced[nMover].SetVeloItp := stPointerAddresses[nMover].SetVeloItpPointer^;
END_FOR
END_METHOD

METHOD GetActHwPosModuloPointer : POINTER TO DINT
VAR_INPUT
	ControllerOID : OTCID;
END_VAR
VAR
	ipComObject			: ITcWatchSource;
	oidActHwPosModulo	: OTCID := 16#A0000010;
	sizeData			: UDINT;
	adrData 			: PVOID; 
END_VAR

nErrorID := FW_ObjMgr_GetObjectInstance(	oid		:=	ControllerOID, 
											iid		:=	TC_GLOBAL_IID_LIST.IID_ITcWatchSource, 
											pipUnk 	:= ADR(ipComObject));


																				
IF ipComObject <> 0 THEN
	
	sizeData := SIZEOF(GetActHwPosModuloPointer);
	adrData := ADR(GetActHwPosModuloPointer);

	nErrorID := ipComObject.InterpretGroupOffsetLength( 	indexOffset := oidActHwPosModulo ,
															cbLength 	:= sizeData,
															ppData 		:= adrData);
	ipComObject.TcRelease();	
	ipComObject := 0;													
														
												
END_IF
END_METHOD

METHOD GetActPosErrorPointer : POINTER TO LREAL
VAR_INPUT
	ControllerOID : OTCID;
END_VAR
VAR
	ipComObject			: ITcWatchSource;
	oidActPosError		: OTCID := 16#A0000018;
	sizeData			: UDINT;
	adrData 			: PVOID; 
END_VAR

nErrorID := FW_ObjMgr_GetObjectInstance(	oid		:=	ControllerOID, 
											iid		:=	TC_GLOBAL_IID_LIST.IID_ITcWatchSource, 
											pipUnk 	:= ADR(ipComObject));


																				
IF ipComObject <> 0 THEN
	
	sizeData := SIZEOF(GetActPosErrorPointer);
	adrData := ADR(GetActPosErrorPointer);

	nErrorID := ipComObject.InterpretGroupOffsetLength( 	indexOffset := oidActPosError ,
															cbLength 	:= sizeData,
															ppData 		:= adrData);
	ipComObject.TcRelease();	
	ipComObject := 0;													
														
												
END_IF
END_METHOD

METHOD GetActVeloPointer : POINTER TO LREAL
VAR_INPUT
	ControllerOID : OTCID;
END_VAR
VAR
	ipComObject			: ITcWatchSource;
	oidActVelo	: OTCID := 16#A0000008;
	sizeData			: UDINT;
	adrData 			: PVOID; 
END_VAR

nErrorID := FW_ObjMgr_GetObjectInstance(	oid		:=	ControllerOID, 
											iid		:=	TC_GLOBAL_IID_LIST.IID_ITcWatchSource, 
											pipUnk 	:= ADR(ipComObject));


																				
IF ipComObject <> 0 THEN
	
	sizeData := SIZEOF(GetActVeloPointer);
	adrData := ADR(GetActVeloPointer);

	nErrorID := ipComObject.InterpretGroupOffsetLength( 	indexOffset := oidActVelo ,
															cbLength 	:= sizeData,
															ppData 		:= adrData);
	ipComObject.TcRelease();	
	ipComObject := 0;													
														
												
END_IF
END_METHOD

METHOD GetSetAccItpPointer : POINTER TO LREAL
VAR_INPUT
	ControllerOID : OTCID;
END_VAR
VAR
	ipComObject			: ITcWatchSource;
	oidSetAccItp		: OTCID := 16#A0000038;
	sizeData			: UDINT;
	adrData 			: PVOID; 
END_VAR

nErrorID := FW_ObjMgr_GetObjectInstance(	oid		:=	ControllerOID, 
											iid		:=	TC_GLOBAL_IID_LIST.IID_ITcWatchSource, 
											pipUnk 	:= ADR(ipComObject));


																				
IF ipComObject <> 0 THEN
	
	sizeData := SIZEOF(GetSetAccItpPointer);
	adrData := ADR(GetSetAccItpPointer);

	nErrorID := ipComObject.InterpretGroupOffsetLength( 	indexOffset := oidSetAccItp ,
															cbLength 	:= sizeData,
															ppData 		:= adrData);
	ipComObject.TcRelease();	
	ipComObject := 0;													
														
												
END_IF
END_METHOD

METHOD GetSetCurrentPointer : POINTER TO LREAL
VAR_INPUT
	ControllerOID : OTCID;
END_VAR
VAR
	ipComObject			: ITcWatchSource;
	oidSetCurrent 		: OTCID := 16#A0000048;
	sizeData			: UDINT;
	adrData 			: PVOID; 
END_VAR

nErrorID := FW_ObjMgr_GetObjectInstance(	oid		:=	ControllerOID, 
											iid		:=	TC_GLOBAL_IID_LIST.IID_ITcWatchSource, 
											pipUnk 	:= ADR(ipComObject));


																				
IF ipComObject <> 0 THEN
	
	sizeData := SIZEOF(GetSetCurrentPointer);
	adrData := ADR(GetSetCurrentPointer);

	nErrorID := ipComObject.InterpretGroupOffsetLength( 	indexOffset := oidSetCurrent ,
															cbLength 	:= sizeData,
															ppData 		:= adrData);
	ipComObject.TcRelease();	
	ipComObject := 0;													
														
												
END_IF
END_METHOD

METHOD GetSetVeloItpPointer : POINTER TO LREAL
VAR_INPUT
	ControllerOID : OTCID;
END_VAR
VAR
	ipComObject			: ITcWatchSource;
	oidSetVeloItp	: OTCID := 16#A0000030;
	sizeData			: UDINT;
	adrData 			: PVOID; 
END_VAR

nErrorID := FW_ObjMgr_GetObjectInstance(	oid		:=	ControllerOID, 
											iid		:=	TC_GLOBAL_IID_LIST.IID_ITcWatchSource, 
											pipUnk 	:= ADR(ipComObject));


																				
IF ipComObject <> 0 THEN
	
	sizeData := SIZEOF(GetSetVeloItpPointer);
	adrData := ADR(GetSetVeloItpPointer);

	nErrorID := ipComObject.InterpretGroupOffsetLength( 	indexOffset := oidSetVeloItp ,
															cbLength 	:= sizeData,
															ppData 		:= adrData);
	ipComObject.TcRelease();	
	ipComObject := 0;													
														
												
END_IF
END_METHOD

METHOD Init : BOOL
VAR_INPUT
END_VAR

VAR_INST
	nState : INT; 
	i : INT; 
	
END_VAR


CASE nState OF 
	
	0: //Get Controller OID 
	
		FOR nMover:= 1 TO nNumOfMovers DO
			
			ControllerOID[nMover] := fbXtsEnv.XpuTcIo(1).MoverTcIo(nMover).GetMoverControllerOid();
				
			stPointerAddresses[nMover].ActHwPosModuloPointer := GetActHwPosModuloPointer(ControllerOID[nMover]);
			stPointerAddresses[nMover].SetVeloItpPointer := GetSetVeloItpPointer(ControllerOID[nMover]);
			stPointerAddresses[nMover].ActVeloPointer := GetActVeloPointer(ControllerOID[nMover]);
			stPointerAddresses[nMover].SetAccItpPointer := GetSetAccItpPointer(ControllerOID[nMover]);
			stPointerAddresses[nMover].ActPosErrorPointer := GetActPosErrorPointer(ControllerOID[nMover]);
			stPointerAddresses[nMover].SetCurrentPointer := GetSetCurrentPointer(ControllerOID[nMover]); 
		
		END_FOR 
	
		nState:= 100; 
		

	100: 
		Init:= TRUE; 
		nState:= 0;

END_CASE
END_METHOD

END_FUNCTION_BLOCK
